TYPE ST_EL6631 :
STRUCT
	bCurrentValueInvalid	: BOOL;
	bCurrentValueUnerRange	: BOOL;
	bCurrentValueOverRange	: BOOL;
	bWarningStatus			: BOOL;
	bErrorStatus			: BOOL;
	iCurrentValue			: DINT;
	iPnIoBoxState			: UINT;
END_STRUCT
END_TYPE

(* stored: Version 1.1.0.1, ProductVersion 3.1.4024.15
   DUT ST_EL6631: Id {af35106f-c497-4e76-9a22-898e3602b328} *)
